FUNCTION_BLOCK McWriteParameter EXTENDS BaseMcProcess
VAR_INPUT
	///Arguments to be set, before writing do_request TRUE
	{attribute 'OPC.UA.DA' := '1'}
	set: McWriteParameterArgs;
END_VAR
VAR_OUTPUT
	///Arguments in use by the process, if do_request was accepted
	{attribute 'OPC.UA.DA' := '1'}
	{attribute 'OPC.UA.DA.Access' := '1'}
	get: McWriteParameterArgs;
END_VAR
VAR_IN_OUT
END_VAR
VAR
END_VAR

IF do_request THEN
    do_request_result := request(
    parameterNumber := set.parameterNumber,
    value := set.value);
    do_request := FALSE;
END_IF;
SUPER^();

{attribute 'TcRpcEnable' := '1'}
METHOD start
VAR_INPUT
	///Number of the parameter
	parameterNumber: INT;
	///Value to write
	value: LREAL;
END_VAR
VAR_OUTPUT
END_VAR
VAR_IN_OUT
END_VAR
VAR
END_VAR
THIS^.get.parameterNumber := parameterNumber;
THIS^.get.value := value;
THIS^.statuses.busyStatus( isBusy := TRUE );
THIS^.statuses.healthStatus( isGood := TRUE );
END_METHOD

{attribute 'TcRpcEnable' := '1'}
METHOD request : RequestResults
VAR_INPUT
	///Number of the parameter
	parameterNumber: INT;
	///Value to write
	value: LREAL;
END_VAR
VAR_OUTPUT
END_VAR
VAR_IN_OUT
END_VAR
VAR
END_VAR
IF THIS^.statuses.enabledStatus.enabled THEN
    THIS^.start(
        parameterNumber := parameterNumber,
        value := value);
    request := RequestResults.ACCEPTED;
ELSE
    request := RequestResults.REJECTED;
END_IF;
END_METHOD

END_FUNCTION_BLOCK

(* stored: Version 1.1.0.1, ProductVersion 3.1.4019.2
   POU McWriteParameter: Id {c483aba3-c65a-4c09-a0aa-1628956f7f4b}, SpecialFunc None
   Method start: Id {ae56391c-fa45-4ef7-ad3e-1199162ac4dd}
   Method request: Id {fb90fc77-7e04-4f4b-8be6-89cb1b38a2dc} *)
